FUNCTION_BLOCK VAV_MDL (* Variable Air Valve Model *)
  (* Standard: 61499-1; Classification: Simulation; ApplicationDomain: HVAC; Function: Variable Air Valve *)
  (* Version 0.1, 2006-05-01, JHC, Holobloc Inc, Changed FV to FD. *)
  (* Version 0.0, 2006-04-10, JHC, Holobloc Inc *)
  (* Compiler header: package fb.rt.hvac; import fb.rt.mva.*; *)
  (* Compiler Java Sun JDK 1.5.0 *)
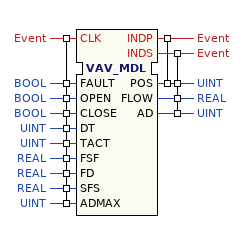
  EVENT_INPUT
    CLK WITH FAULT, OPEN, CLOSE, DT, TACT, FSF, FD, SFS, ADMAX; (* External Clock Event *)
  END_EVENT
  EVENT_OUTPUT
    INDP WITH POS; (* POS changed *)
    INDS WITH POS, FLOW, AD; (* Sensor value changed (always follows CLK) *)
  END_EVENT
  VAR_INPUT
    FAULT : BOOL; (* 0=Enable,1=Simulate Fault *)
    OPEN : BOOL; (* Open Damper *)
    CLOSE : BOOL; (* Close Damper *)
    DT : UINT := 10; (* Clock period, sec *)
    TACT : UINT := 95; (* Damper actuation time, sec *)
    FSF : REAL := 1000.0; (* Air Flow at Damper Full Open, CFM *)
    FD : REAL; (* Maximum random flow deviation in CFM *)
    SFS : REAL := 1000.0; (* Air Flow at Sensor Full Scale, CFM *)
    ADMAX : UINT := 4096; (* Maximum Flow Sensor A/D converter value + 1, default is 12 bits *)
  END_VAR
  VAR_OUTPUT
    POS : UINT; (* Damper position, 0..100% open *)
    FLOW : REAL; (* Air flow, CFM *)
    AD : UINT; (* Flow sensor A/D converter value *)
  END_VAR
  FBS
    DAMPER : MECH2_MDL;
    PRE : VAV_PRE;
    POST : VAV_POST;
    SPLT : E_SPLIT; (* Ensure CNF output *)
  END_FBS
  EVENT_CONNECTIONS
    CLK TO PRE.CLK;
    POST.CNF TO INDS;
    PRE.CNF TO SPLT.EI;
    SPLT.EO1 TO DAMPER.CLK;
    SPLT.EO2 TO POST.CLK;
    DAMPER.INDP TO INDP;
  END_CONNECTIONS
  DATA_CONNECTIONS
    FAULT TO DAMPER.FAULT;
    OPEN TO DAMPER.FWD;
    CLOSE TO DAMPER.REV;
    DAMPER.POS TO POS;
    DT TO PRE.DT;
    TACT TO PRE.TACT;
    PRE.V TO DAMPER.VF;
    PRE.V TO DAMPER.VR;
    DAMPER.POS TO POST.POS;
    SFS TO POST.SFS;
    FSF TO POST.FSF;
    FD TO POST.FD;
    ADMAX TO POST.ADMAX;
    POST.FLOW TO FLOW;
    POST.AD TO AD;
  END_CONNECTIONS
END_FUNCTION_BLOCK
